(* Logix 5000 project; controller DC01 vendor 1 type 14 code 165 rev 32.12; software revision 32.04; part 13 of 13 *)
(* tags used below, declared in another part *)
   ASSY_COMS_com_status : DINT;   // DC01 Bldg Ethernet Communications To Data Center Status Monitor
   clock_current_string : STRING[13];
   Clock_Min_Pulse : BOOL;
   Clock_Set_Routine : PA_WallClock_UDDT;
   DateTime_Update : BOOL;
   DayOfWeek : DINT;
   DC1_clock_sync : DINT[10];
   DC1_OPCFault : BOOL;
   DC1_OPCWatchDog : BOOL;
   DC1_to_LN01_Messages : DINT[20];
   DC1_to_LN02_Messages : DINT[20];
   DC1_to_LN03_Messages : DINT[20];
   DC1_to_LN04_Messages : DINT[20];
   ENET_COMMS_OK : BOOL;   // DC01 Ethernet Building Network Comms Good
   IGN_DateTime_Record_Current : STRING;
   IGN_Day : DINT;
   IGN_DayPrev : DINT;
   IGN_DayString : STRING;
   IGN_Hour : DINT;
   IGN_HourString : STRING;
   IGN_Minute : DINT;
   IGN_MinuteString : STRING;
   IGN_Month : DINT;
   IGN_MonthString : STRING;
   IGN_Second : DINT;
   IGN_SecondString : STRING;
   IGN_Year : DINT;
   IGN_YearString : STRING;
   LN01_Schedule : UDT_Current_Status;
   LN02_Schedule : UDT_Current_Status;
   LN03_Schedule : UDT_Current_Status;
   LN04_MainLine_MSG_Out : MESSAGE;
   LN04_Schedule : UDT_Current_Status;
   LN04_Theoretical_Units_Counter : COUNTER;
   test : BOOL;
   Test_Result : DINT;
   TestDateTime : DINT;
   TMR_COMMS : TIMER;
(* LN04, continued *)

ROUTINE R04_DataToLines   (* ladder *)
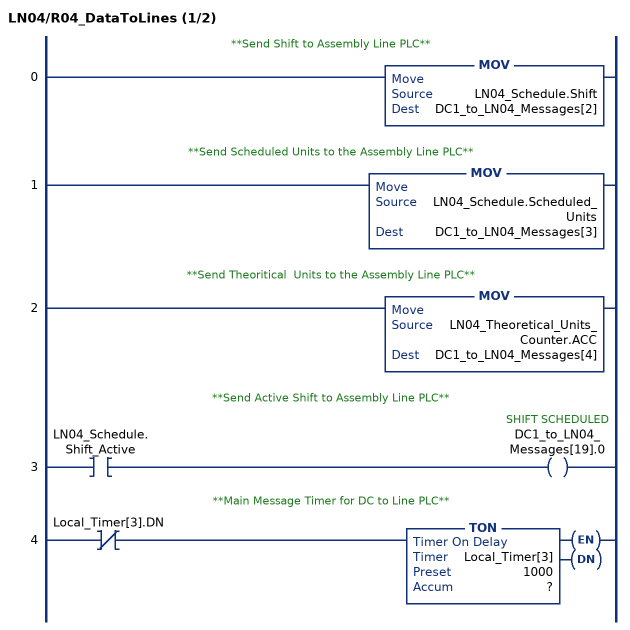
   // **Send Shift to Assembly Line PLC**
   0: MOV(LN04_Schedule.Shift,DC1_to_LN04_Messages[2]);
   // **Send Scheduled Units to the Assembly Line PLC**
   1: MOV(LN04_Schedule.Scheduled_Units,DC1_to_LN04_Messages[3]);
   // **Send Theoritical  Units to the Assembly Line PLC**
   2: MOV(LN04_Theoretical_Units_Counter.ACC,DC1_to_LN04_Messages[4]);
   // **Send Active Shift to Assembly Line PLC**
   3: XIC(LN04_Schedule.Shift_Active)OTE(DC1_to_LN04_Messages[19].0);
   // **Main Message Timer for DC to Line PLC**
   4: XIO(Local_Timer[3].DN)TON(Local_Timer[3],?,?);
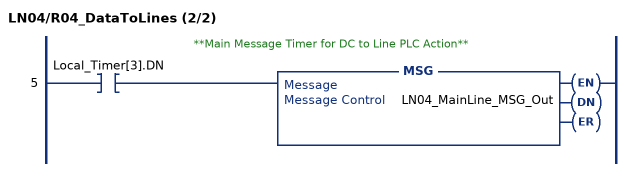
   // **Main Message Timer for DC to Line PLC Action**
   5: XIC(Local_Timer[3].DN)MSG(LN04_MainLine_MSG_Out);
END_ROUTINE
END_PROGRAM

PROGRAM MainProgram   (* main routine MainRoutine *)
VAR
   Array_Track : DINT := 8;
   Clock_Current : DINT[40] := ([0] := 2023, [1] := 5, [2] := 8, [3] := 7, [4] := 55, [5] := 22, [6] := 95622, [10] := 2023, [11] := 5, [12] := 8, [13] := 7, [14] := 55, [15] := 22, [16] := 95622);
   DOW_Century : DINT := 20;   // Century or upper two digits from the year
   DOW_Day : DINT := 7;   // Day of the Month 1-31
   DOW_InputDate : DateTime_Type := (Year := 2023, Month := 5, Day := 8, Hour := 13, Minute := 47, Second := 35, Microseconds := 331852);
   DOW_Month : DINT := 3;   // Month 1 = March, 10=december, 11=Jan and 12=Feb
   DOW_Output : DINT;   // Day of Week 0 = Sun, 1=Mon, 2=Tues, 3=Wed, 4=Thur, 5=Fri, 6=Sat
   DOW_Temp00 : REAL := 20.23;   // Intermediate Math Value
   DOW_Temp01 : REAL := 7.7999997;   // Intermediate Math Value
   DOW_Temp02 : REAL := 7.600001;   // Intermediate Math Value
   DOW_Temp03 : DINT := 7;   // Intermediate Math Value
   DOW_Temp04 : DINT := 40;   // Intermediate Math Value
   DOW_Temp05 : REAL := 5.75;   // Intermediate Math Value
   DOW_Temp06 : DINT := 5;   // Intermediate Math Value
   DOW_Temp07 : REAL := 5.0;   // Intermediate Math Value
   DOW_Temp08 : DINT := 5;   // Intermediate Math Value
   DOW_Temp09 : REAL := 14.0;   // Intermediate Math Value
   DOW_Temp10 : REAL := -26.0;   // Intermediate Math Value
   DOW_Temp11 : REAL := -3.0;   // Intermediate Math Value
   DOW_Temp12 : REAL := 2.0;   // Intermediate Math Value
   DOW_Temp13 : REAL := 7.0;   // Intermediate Math Value
   DOW_Temp14 : REAL;   // Intermediate Math Value
   DOW_Temp15 : REAL;   // Intermediate Math Value
   DOW_Year : DINT := 23;   // Year within the century or last two digits in year
   Local_Bool : BOOL[32];
   Local_DATETIME : DINT[10] := ([0] := 2023, [1] := 5, [2] := 8, [3] := 7, [4] := 55, [5] := 24, [6] := 214453);
   Local_DateTimeSet : DINT[20] := ([0] := 2023, [1] := 5, [2] := 8, [3] := 7, [4] := 55, [5] := 22);
   Local_Timer : TIMER[5] := ([0].PRE := 6500, [0].ACC := 6500, [0].EN := 1, [0].DN := 1, [1].PRE := 6500);
   ONS : BOOL[32] := ([0] := 1);
   OPCFaultDateTime : STRING[10] := ([0] := '2022', [1] := '11', [2] := '25', [3] := '19', [4] := '54', [5] := '55');
   Previous_Minute : DINT := 55;
   str_DateTimeStamp : STRING[10] := ([0] := '2023', [1] := '5', [2] := '8', [3] := '7', [4] := '55', [5] := '24', [6] := '626169');
END_VAR

ROUTINE CLOCK_SET   (* ladder *)
// ROUTINE TO SET CLOCK
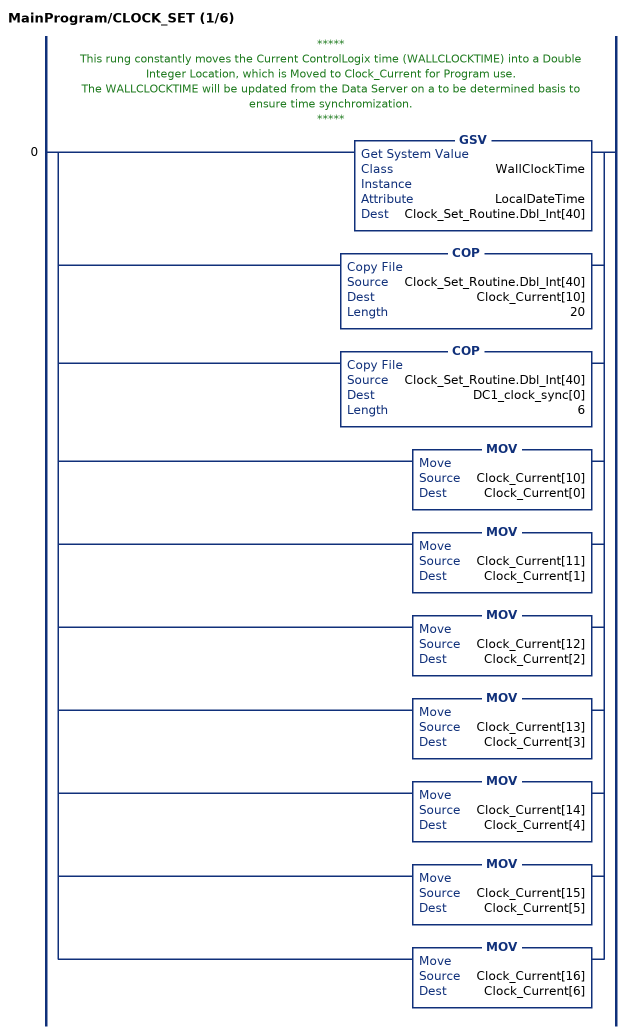
   // *****
   // This rung constantly moves the Current ControlLogix time (WALLCLOCKTIME) into a Double Integer Location, which is Moved to Clock_Current for Program use.
   // The WALLCLOCKTIME will be updated from the Data Server on a to be determined basis to ensure time synchromization.
   // *****
   0: [GSV(WallClockTime,,LocalDateTime,Clock_Set_Routine.Dbl_Int[40]) ,COP(Clock_Set_Routine.Dbl_Int[40],Clock_Current[10],20) ,COP(Clock_Set_Routine.Dbl_Int[40],DC1_clock_sync[0],6) ,MOV(Clock_Current[10],Clock_Current[0]) ,MOV(Clock_Current[11],Clock_Current[1]) ,MOV(Clock_Current[12],Clock_Current[2]) ,MOV(Clock_Current[13],Clock_Current[3]) ,MOV(Clock_Current[14],Clock_Current[4]) ,MOV(Clock_Current[15],Clock_Current[5]) ,MOV(Clock_Current[16],Clock_Current[6]) ];
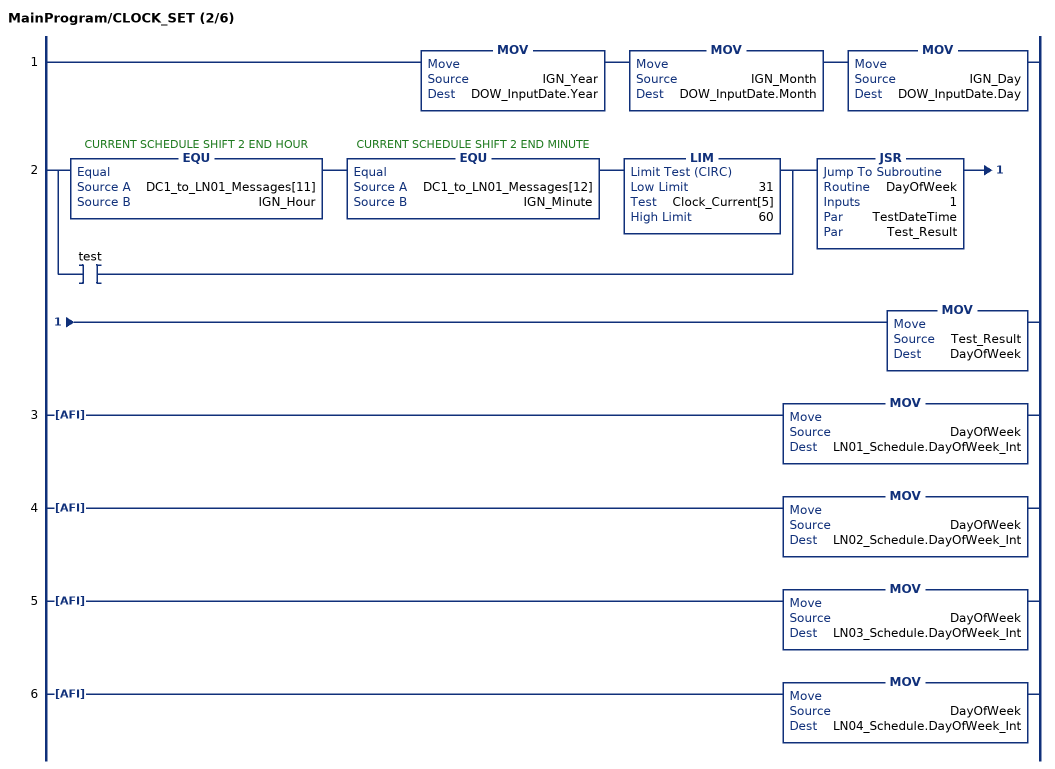
   1: MOV(IGN_Year,DOW_InputDate.Year)MOV(IGN_Month,DOW_InputDate.Month)MOV(IGN_Day,DOW_InputDate.Day);
   2: [EQU(DC1_to_LN01_Messages[11],IGN_Hour) EQU(DC1_to_LN01_Messages[12],IGN_Minute) LIM(31,Clock_Current[5],60) ,XIC(test) ]JSR(DayOfWeek,1,TestDateTime,Test_Result)MOV(Test_Result,DayOfWeek);
   3: AFI()MOV(DayOfWeek,LN01_Schedule.DayOfWeek_Int);
   4: AFI()MOV(DayOfWeek,LN02_Schedule.DayOfWeek_Int);
   5: AFI()MOV(DayOfWeek,LN03_Schedule.DayOfWeek_Int);
   6: AFI()MOV(DayOfWeek,LN04_Schedule.DayOfWeek_Int);
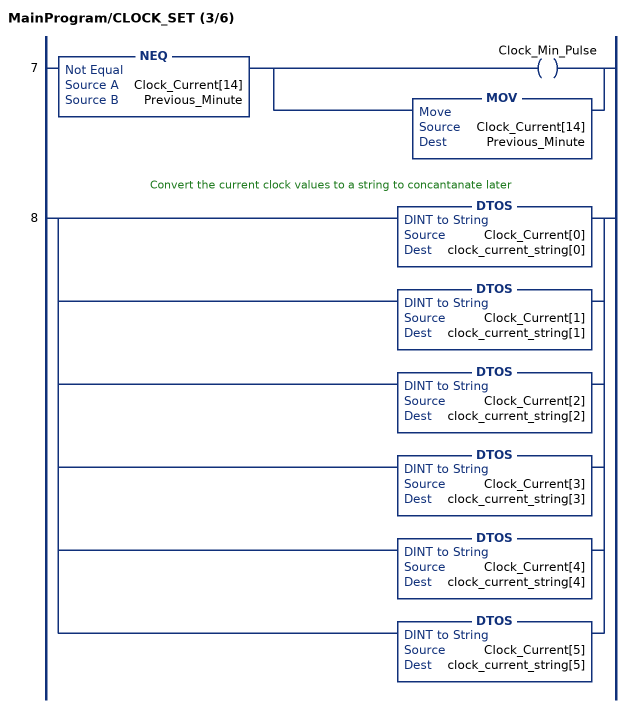
   7: NEQ(Clock_Current[14],Previous_Minute)[OTE(Clock_Min_Pulse) ,MOV(Clock_Current[14],Previous_Minute) ];
   // Convert the current clock values to a string to concantanate later
   8: [DTOS(Clock_Current[0],clock_current_string[0]) ,DTOS(Clock_Current[1],clock_current_string[1]) ,DTOS(Clock_Current[2],clock_current_string[2]) ,DTOS(Clock_Current[3],clock_current_string[3]) ,DTOS(Clock_Current[4],clock_current_string[4]) ,DTOS(Clock_Current[5],clock_current_string[5]) ];
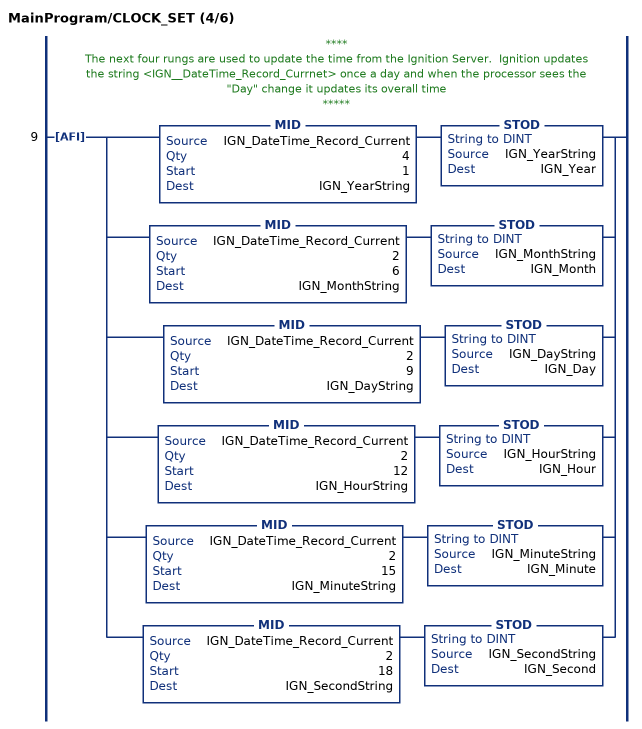
   // ****
   // The next four rungs are used to update the time from the Ignition Server.  Ignition updates the string <IGN__DateTime_Record_Currnet> once a day and when the processor sees the "Day" change it updates its overall time
   // *****
   9: AFI()[MID(IGN_DateTime_Record_Current,4,1,IGN_YearString) STOD(IGN_YearString,IGN_Year) ,MID(IGN_DateTime_Record_Current,2,6,IGN_MonthString) STOD(IGN_MonthString,IGN_Month) ,MID(IGN_DateTime_Record_Current,2,9,IGN_DayString) STOD(IGN_DayString,IGN_Day) ,MID(IGN_DateTime_Record_Current,2,12,IGN_HourString) STOD(IGN_HourString,IGN_Hour) ,MID(IGN_DateTime_Record_Current,2,15,IGN_MinuteString) STOD(IGN_MinuteString,IGN_Minute) ,MID(IGN_DateTime_Record_Current,2,18,IGN_SecondString) STOD(IGN_SecondString,IGN_Second) ];
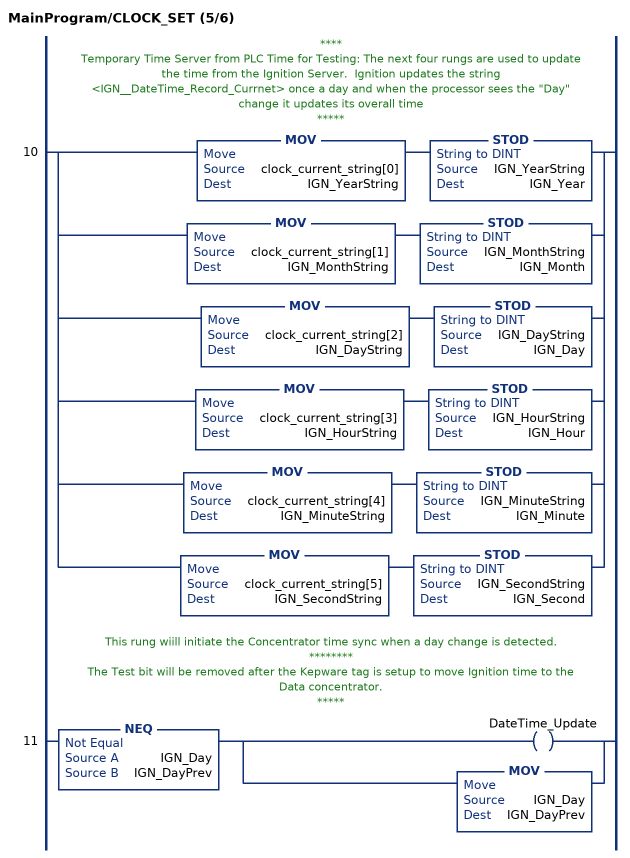
   // ****
   // Temporary Time Server from PLC Time for Testing: The next four rungs are used to update the time from the Ignition Server.  Ignition updates the string <IGN__DateTime_Record_Currnet> once a day and when the processor sees the "Day" change it updates its overall time
   // *****
   10: [MOV(clock_current_string[0],IGN_YearString) STOD(IGN_YearString,IGN_Year) ,MOV(clock_current_string[1],IGN_MonthString) STOD(IGN_MonthString,IGN_Month) ,MOV(clock_current_string[2],IGN_DayString) STOD(IGN_DayString,IGN_Day) ,MOV(clock_current_string[3],IGN_HourString) STOD(IGN_HourString,IGN_Hour) ,MOV(clock_current_string[4],IGN_MinuteString) STOD(IGN_MinuteString,IGN_Minute) ,MOV(clock_current_string[5],IGN_SecondString) STOD(IGN_SecondString,IGN_Second) ];
   // This rung wiill initiate the Concentrator time sync when a day change is detected.
   // ********
   // The Test bit will be removed after the Kepware tag is setup to move Ignition time to the Data concentrator.
   // *****
   11: NEQ(IGN_Day,IGN_DayPrev)[OTE(DateTime_Update) ,MOV(IGN_Day,IGN_DayPrev) ];
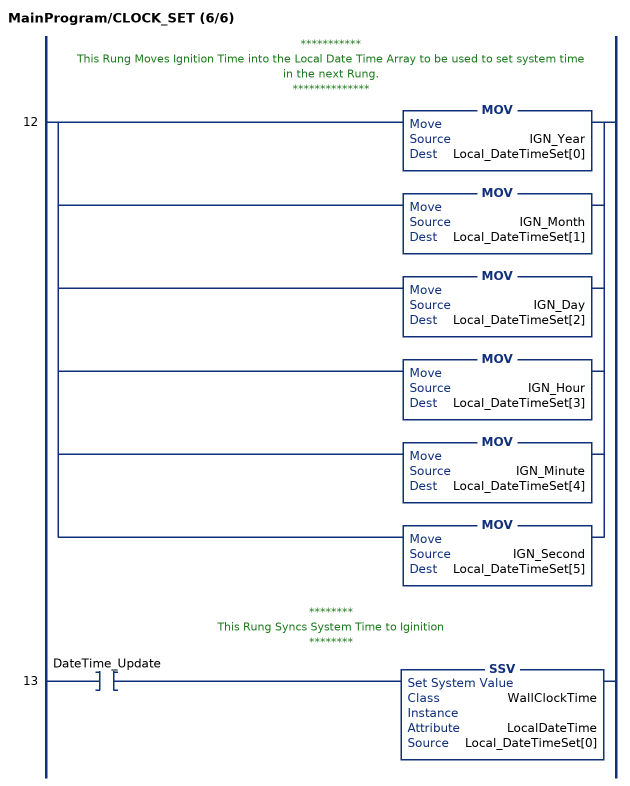
   // ***********
   // This Rung Moves Ignition Time into the Local Date Time Array to be used to set system time in the next Rung.
   // **************
   12: [MOV(IGN_Year,Local_DateTimeSet[0]) ,MOV(IGN_Month,Local_DateTimeSet[1]) ,MOV(IGN_Day,Local_DateTimeSet[2]) ,MOV(IGN_Hour,Local_DateTimeSet[3]) ,MOV(IGN_Minute,Local_DateTimeSet[4]) ,MOV(IGN_Second,Local_DateTimeSet[5]) ];
   // ********
   // This Rung Syncs System Time to Iginition
   // ********
   13: XIC(DateTime_Update)SSV(WallClockTime,,LocalDateTime,Local_DateTimeSet[0]);
END_ROUTINE

ROUTINE DayOfWeek   (* ladder *)
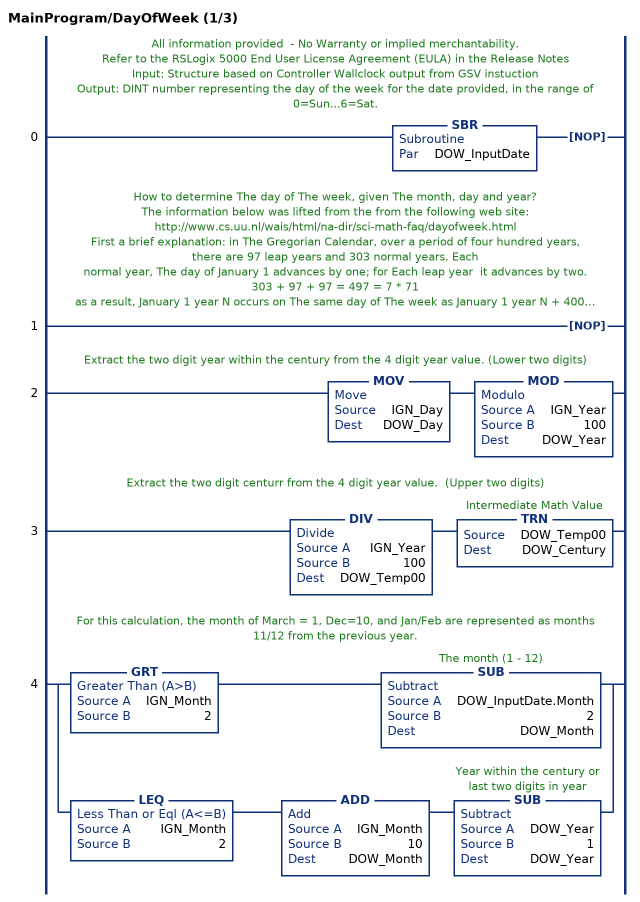
   // All information provided  - No Warranty or implied merchantability.
   // Refer to the RSLogix 5000 End User License Agreement (EULA) in the Release Notes
   // Input: Structure based on Controller Wallclock output from GSV instuction
   // Output: DINT number representing the day of the week for the date provided, in the range of 0=Sun...6=Sat.
   0: SBR(DOW_InputDate)NOP();
   // How to determine The day of The week, given The month, day and year?
   // The information below was lifted from the from the following web site: http://www.cs.uu.nl/wais/html/na-dir/sci-math-faq/dayofweek.html
   //    First a brief explanation: in The Gregorian Calendar, over a period of four hundred years, there are 97 leap years and 303 normal years. Each
   //  normal year, The day of January 1 advances by one; for Each leap year  it advances by two.
   //    303 + 97 + 97 = 497 = 7 * 71
   //    as a result, January 1 year N occurs on The same day of The week as January 1 year N + 400. Because The leap year pattern also recurs with a four hundred year cycle, a simple table of four hundred elements, and single modulus, suffices to determine The day of The week (in The
   //    Gregorian Calendar), and does it much faster than all The other algorithms proposed. also, Each element takes (in principle) only three bits; The entire table thus takes only 1200 bits; on many computers this will be less than The instructions to do all The complicated calculations proposed or The other algorithms.
   //    Incidental Note: Because 7 does not Divide 400, January 1 occurs more frequently on some days than others! Trick your friends! in a cycle of 400 years, January 1 and March 1 occur on The following days with The following frequencies:
   //            Sun      Mon     Tue     Wed     Thu     Fri     Sat
   //     Jan 1: 58       56      58      57      57      58      56
   //     Mar 1: 58       56      58      56      58      57      57
   //    Of interest is that (contrary to most initial guesses) The occurrence is not maximally flat.
   // In The Mathematical Gazette, vol. 53,, pp.127-129, it is shown that The 13th of The month is more likely to be a Friday than any other day.The author is a 13 year old S.R.Baxter.
   //    The Gregorian Calendar was introduced in 1582 in parts of Europe; it was adopted in 1752 in Great Britain and its colonies, and on various dates in other countries. it replaced The Julian Calendar which has a four-year cycle of leap years; after four years January 1 has advanced by five days. Since 5 is relatively prime to 7, a table of 4 * 7 = 28 elements is necessary for The Julian Calendar.
   //    there is still a 3 day over 10,000 years error which The Gregorian Calendar does not take into account. At some Time such a correction will have to be done but your software will probably not last that long!
   //    Here is a standard method suitable for mental computation:
   //     1. take The last two digits of The year.
   //     2. Divide by 4, discarding any fraction.
   //     3. Add The day of The month.
   //     4. Add The month'S key value: JFM AMJ JAS OND 144 025 036 146
   //     5. Subtract 1 for January or February of a leap year.
   //     6. For a Gregorian Date, Add 0 for 1900'S, 6 for 2000'S, 4 for 1700'S, 2 for 1800'S; for other years, Add or Subtract multiples of 400.
   //     7. For a Julian Date, Add 1 for 1700'S, and 1 for every additional century you go back.
   //     8. Add The last two digits of The year.
   //     9. Divide by 7 and take The remainder.
   //    Now 1 is Sunday, The First day of The week, 2 is Monday, and so on.
   //    The following formula, which is for The Gregorian Calendar only, may be more convenient for computer programming. Note that in some programming languages The remainder operation can yield a negative result if given a negative operand, so mod 7 may not translate to a simple remainder.
   //    W = (k + floor(2.6m - 0.2) - 2C + Y + floor(Y/4) + floor(C/4)) mod 7
   //    where floor() denotes The integer floor function [This is TRN() in Logix],
   // k is day (1 to 31)
   //  m is month (1 = March, ..., 10 = December, 11 = Jan, 12 = Feb) Treat Jan & Feb as months of The preceding year
   //    C is century (1987 has C = 19)
   //    Y is year (1987 has Y = 87 except Y = 86 for Jan & Feb)
   //    W is week day (0 = Sunday, ..., 6 = Saturday)
   //    Here The century and 400 year corrections are built into The formula. The floor(2.6m - 0.2) term relates to The repetitive pattern that The 30-day months show when March is taken as The First month.
   //    The following short C program works for a restricted range, it returns 0 for Monday, 1 for Tuesday, etc.
   // dow(m,d,Y){Y-=m<3;return(Y+Y/4-Y/100+Y/400+[m]+d)%7;}
   //    The program appeared was posted by sakamoto@sm.sony.co.jp (Tomohiko sakamoto) on comp.lang.c on March 10th, 1993.
   //    a good mnemonic rule to help on The computation of The day of The week is as follows. in any given year The following days come on The same day of The week: 4/4, 6/6, 8/8, 10/10, 12/12  to remember The next four, remember that I work from 9-5 At a 7-11 so 9/5, 5/9, 7/11, 11/7 and The last day of Feb.
   //    Even ignoring The pattern over for a period of years this is still useful Since you can generally figure out what day of The week a given Date is  on faster than someone else can look it up with a calender if The calender is not right there. (a useful skill that.)
   //  References:
   //    Winning Ways for your Mathematical plays. Elwyn R. Berlekamp, John H.  Conway, and Richard k. Guy London ; Toronto : Academic Press, 1982.
   //    Mathematical Carnival. Martin Gardner. New York : Knopf, c1975.
   //    Elementary Number Theory and its applications. Kenneth Rosen. Reading,  Mass. ; Don Mills, Ont. : Addison-Wesley Pub. Co., c1993. p. 156.
   //    Michael Keith and Tom Craver. The Ultimate Perpetual Calendar? Journal of Recreational Mathematics, 22:4, pp. 280-282, 19
   1: NOP();
   // Extract the two digit year within the century from the 4 digit year value. (Lower two digits)
   2: MOV(IGN_Day,DOW_Day)MOD(IGN_Year,100,DOW_Year);
   // Extract the two digit centurr from the 4 digit year value.  (Upper two digits)
   3: DIV(IGN_Year,100,DOW_Temp00)TRN(DOW_Temp00,DOW_Century);
   // For this calculation, the month of March = 1, Dec=10, and Jan/Feb are represented as months 11/12 from the previous year.
   4: [GRT(IGN_Month,2) SUB(DOW_InputDate.Month,2,DOW_Month) ,LEQ(IGN_Month,2) ADD(IGN_Month,10,DOW_Month) SUB(DOW_Year,1,DOW_Year) ];
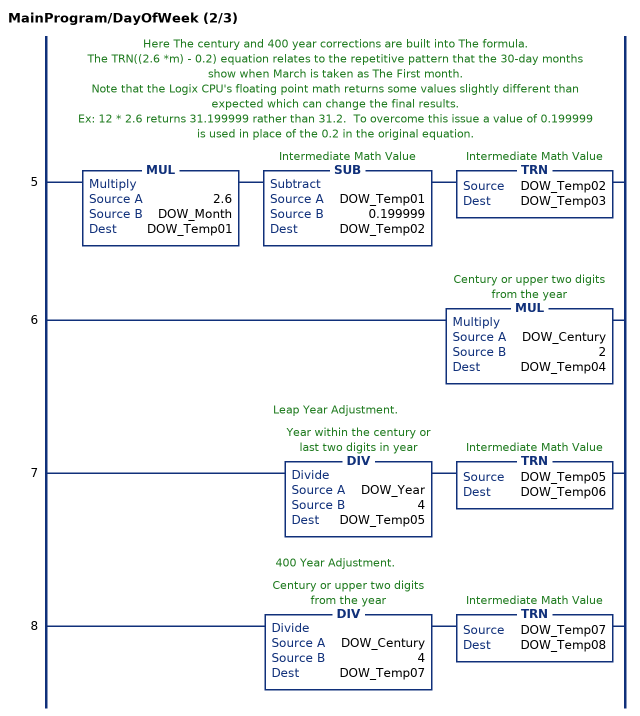
   // Here The century and 400 year corrections are built into The formula.
   // The TRN((2.6 *m) - 0.2) equation relates to the repetitive pattern that the 30-day months show when March is taken as The First month.
   // Note that the Logix CPU's floating point math returns some values slightly different than expected which can change the final results.
   // Ex: 12 * 2.6 returns 31.199999 rather than 31.2.  To overcome this issue a value of 0.199999 is used in place of the 0.2 in the original equation.
   5: MUL(2.6,DOW_Month,DOW_Temp01)SUB(DOW_Temp01,0.199999,DOW_Temp02)TRN(DOW_Temp02,DOW_Temp03);
   6: MUL(DOW_Century,2,DOW_Temp04);
   // Leap Year Adjustment.
   7: DIV(DOW_Year,4,DOW_Temp05)TRN(DOW_Temp05,DOW_Temp06);
   // 400 Year Adjustment.
   8: DIV(DOW_Century,4,DOW_Temp07)TRN(DOW_Temp07,DOW_Temp08);
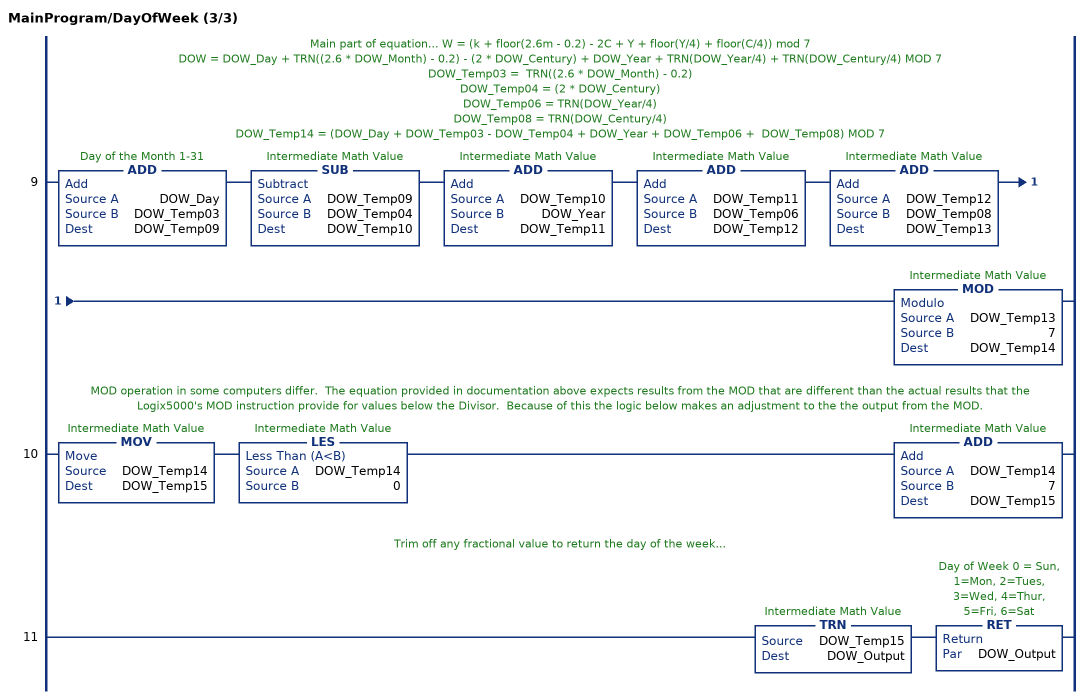
   // Main part of equation... W = (k + floor(2.6m - 0.2) - 2C + Y + floor(Y/4) + floor(C/4)) mod 7
   // DOW = DOW_Day + TRN((2.6 * DOW_Month) - 0.2) - (2 * DOW_Century) + DOW_Year + TRN(DOW_Year/4) + TRN(DOW_Century/4) MOD 7
   // DOW_Temp03 =  TRN((2.6 * DOW_Month) - 0.2)
   // DOW_Temp04 = (2 * DOW_Century)
   // DOW_Temp06 = TRN(DOW_Year/4)
   // DOW_Temp08 = TRN(DOW_Century/4)
   // DOW_Temp14 = (DOW_Day + DOW_Temp03 - DOW_Temp04 + DOW_Year + DOW_Temp06 +  DOW_Temp08) MOD 7
   9: ADD(DOW_Day,DOW_Temp03,DOW_Temp09)SUB(DOW_Temp09,DOW_Temp04,DOW_Temp10)ADD(DOW_Temp10,DOW_Year,DOW_Temp11)ADD(DOW_Temp11,DOW_Temp06,DOW_Temp12)ADD(DOW_Temp12,DOW_Temp08,DOW_Temp13)MOD(DOW_Temp13,7,DOW_Temp14);
   // MOD operation in some computers differ.  The equation provided in documentation above expects results from the MOD that are different than the actual results that the Logix5000's MOD instruction provide for values below the Divisor.  Because of this the logic below makes an adjustment to the the output from the MOD.
   10: MOV(DOW_Temp14,DOW_Temp15)LES(DOW_Temp14,0)ADD(DOW_Temp14,7,DOW_Temp15);
   // Trim off any fractional value to return the day of the week...
   11: TRN(DOW_Temp15,DOW_Output)RET(DOW_Output);
END_ROUTINE

ROUTINE MainRoutine   (* ladder *)
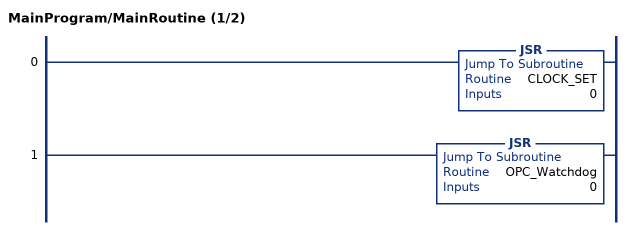
   0: JSR(CLOCK_SET,0);
   1: JSR(OPC_Watchdog,0);
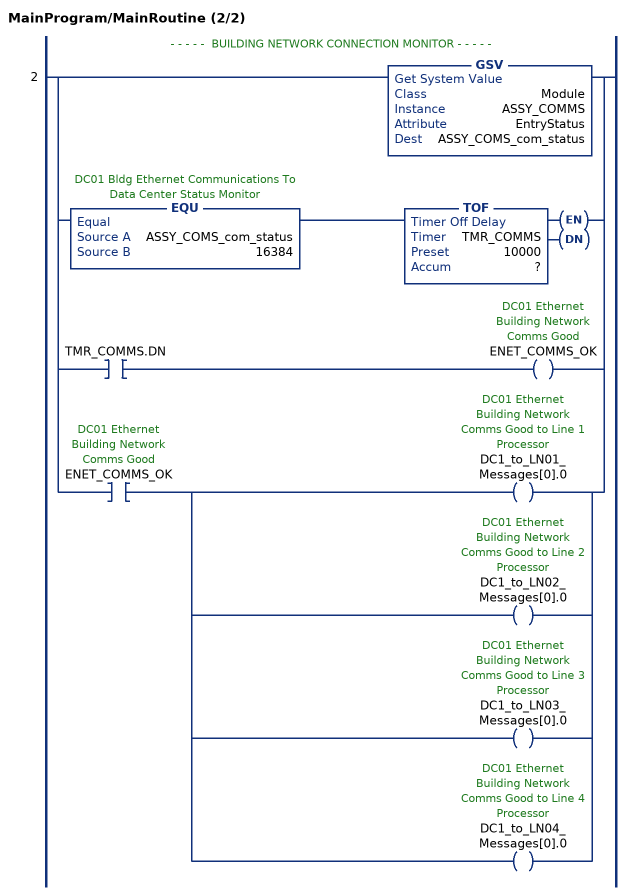
   // - - - - -  BUILDING NETWORK CONNECTION MONITOR - - - - -
   2: [GSV(Module,ASSY_COMMS,EntryStatus,ASSY_COMS_com_status) ,EQU(ASSY_COMS_com_status,16384) TOF(TMR_COMMS,?,?) ,XIC(TMR_COMMS.DN) OTE(ENET_COMMS_OK) ,XIC(ENET_COMMS_OK) [OTE(DC1_to_LN01_Messages[0].0) ,OTE(DC1_to_LN02_Messages[0].0) ,OTE(DC1_to_LN03_Messages[0].0) ,OTE(DC1_to_LN04_Messages[0].0) ] ];
END_ROUTINE

ROUTINE OPC_Watchdog   (* ladder *)
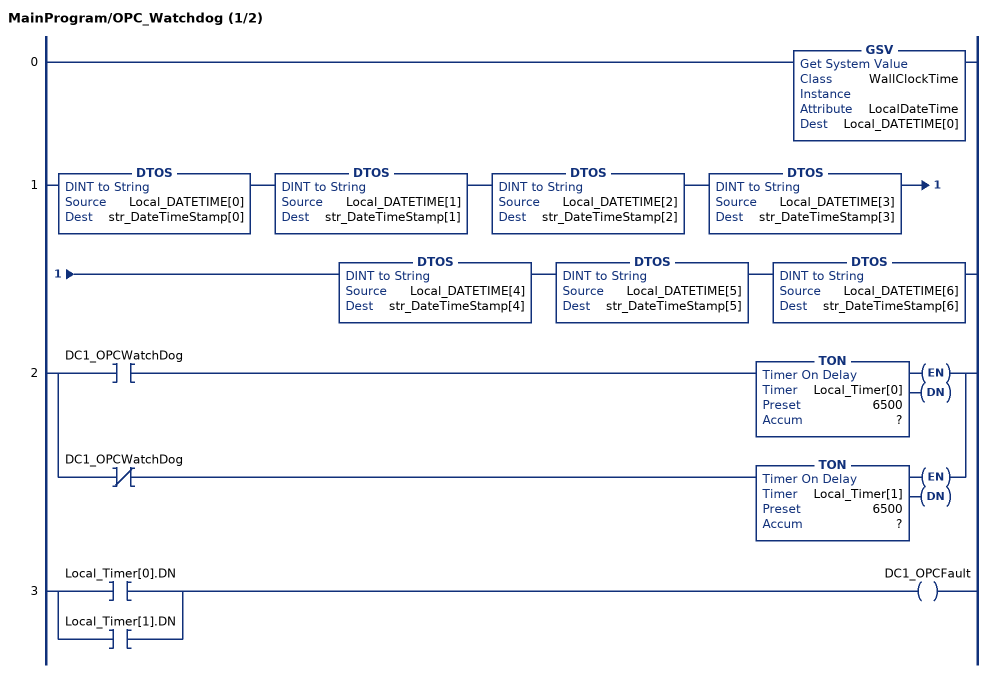
   0: GSV(WallClockTime,,LocalDateTime,Local_DATETIME[0]);
   1: DTOS(Local_DATETIME[0],str_DateTimeStamp[0])DTOS(Local_DATETIME[1],str_DateTimeStamp[1])DTOS(Local_DATETIME[2],str_DateTimeStamp[2])DTOS(Local_DATETIME[3],str_DateTimeStamp[3])DTOS(Local_DATETIME[4],str_DateTimeStamp[4])DTOS(Local_DATETIME[5],str_DateTimeStamp[5])DTOS(Local_DATETIME[6],str_DateTimeStamp[6]);
   2: [XIC(DC1_OPCWatchDog) TON(Local_Timer[0],?,?) ,XIO(DC1_OPCWatchDog) TON(Local_Timer[1],?,?) ];
   3: [XIC(Local_Timer[0].DN) ,XIC(Local_Timer[1].DN) ]OTE(DC1_OPCFault);
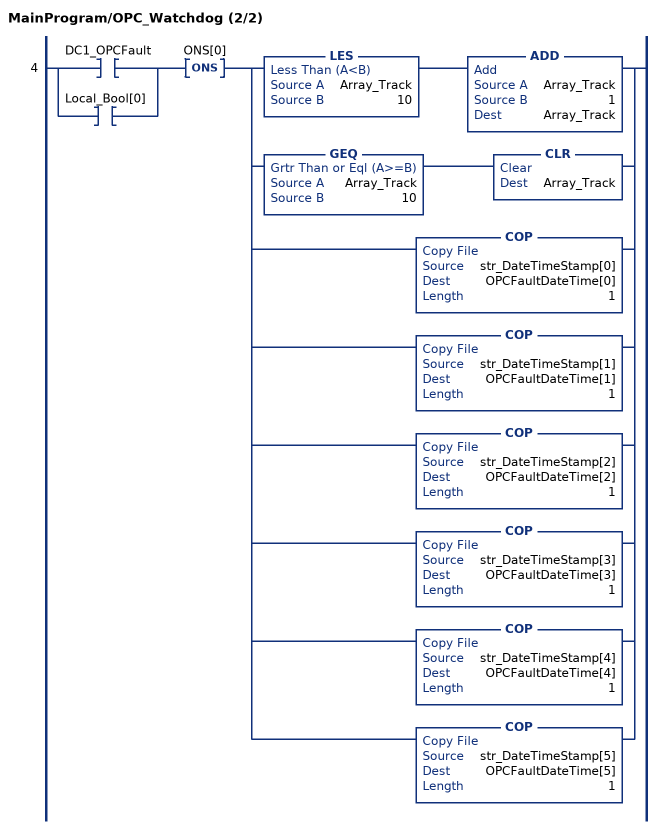
   4: [XIC(DC1_OPCFault) ,XIC(Local_Bool[0]) ]ONS(ONS[0])[LES(Array_Track,10) ADD(Array_Track,1,Array_Track) ,GEQ(Array_Track,10) CLR(Array_Track) ,COP(str_DateTimeStamp[0],OPCFaultDateTime[0],1) ,COP(str_DateTimeStamp[1],OPCFaultDateTime[1],1) ,COP(str_DateTimeStamp[2],OPCFaultDateTime[2],1) ,COP(str_DateTimeStamp[3],OPCFaultDateTime[3],1) ,COP(str_DateTimeStamp[4],OPCFaultDateTime[4],1) ,COP(str_DateTimeStamp[5],OPCFaultDateTime[5],1) ];
END_ROUTINE
END_PROGRAM
